Yaskawa INFORM job: KRIS5(-224_-90).JBI

/JOB
//NAME KRIS5(-224_-90)
//POS
///NPOS 254,254,254,14,0,0
///TOOL 0
///POSTYPE PULSE
///PULSE
C00000=126,-73357,-105376,-18827,72039,-77556
C00001=35778,-73357,-105376,-18827,72039,-77556
C00002=13505,189291,121101,-6814,55937,-83682
C00003=119958,189291,121101,-6814,55937,-83682
C00004=119958,189291,121101,-6814,55937,-83682
C00005=119958,189291,121101,-6814,96257,-82158
C00006=69507,150313,105301,-6814,81918,-83682
C00007=72199,118597,79738,-6814,91004,-83682
C00008=-14837,117754,79738,-6814,76523,-83682
C00009=-41681,102292,47908,-7222,67797,-83732
C00010=-106120,216,-72664,-1265,72875,-87293
C00011=-133015,-103640,-65816,3996,83698,-82063
C00012=-132086,-97485,-64003,4135,58701,-800
C00013=-131334,-97837,-53111,16599,61159,17527
C00014=-132395,-95402,-50215,16816,60857,17080
C00015=-132416,-94549,-48691,16897,60382,16996
C00016=-132416,-94725,-48971,16883,60461,17009
C00017=-132279,-93851,-48637,16827,60667,17094
C00018=-132382,-95256,-50220,16811,60927,17097
C00019=-94304,-90108,-48639,9529,56492,31191
C00020=-93667,-91692,-48976,9441,55822,31379
C00021=-93667,-90817,-47524,9489,55384,31339
C00022=-93667,-90990,-47811,9479,55470,31347
C00023=-93978,-90150,-47514,9528,55751,31249
C00024=-93593,-92158,-49496,9416,55894,31412
C00025=-118370,-114314,-60072,-4758,57984,4074
C00026=-118524,-103625,-49497,-4790,56962,4061
C00027=-114721,-103695,-48891,-5314,56776,5470
C00028=-114721,-102430,-47073,-5343,56310,5496
C00029=-114721,-103093,-48027,-5328,56554,5483
C00030=-114967,-100720,-47370,-5249,57351,5352
C00031=-114746,-103713,-49188,-5301,56945,5454
C00032=-161548,-94752,-46532,1465,58857,-11790
C00033=-161391,-93932,-45538,1444,58664,-11736
C00034=-161391,-92965,-44024,1450,58232,-11741
C00035=-161391,-93332,-44604,1446,58395,-11738
C00036=-160555,-92069,-44187,1319,58776,-11425
C00037=-161970,-95177,-46431,1528,58581,-11948
C00038=-123580,-122537,-67579,3227,57871,938
C00039=-106734,-120076,-67764,3834,76101,81400
C00040=-113343,-108186,-55340,6658,74419,78596
C00041=-116418,-106590,-51558,6363,73154,77529
C00042=-116418,-104744,-48943,6384,72498,77494
C00043=-116380,-105629,-49629,6389,72465,77504
C00044=-116257,-107112,-50007,6421,71928,77514
C00045=-116461,-105924,-51247,6354,73311,77523
C00046=-177893,-84927,-44498,-1145,82347,57715
C00047=-179150,-83983,-43048,-1323,81921,57309
C00048=-179150,-83213,-41718,-1324,81495,57312
C00049=-179506,-83879,-42356,-1373,81537,57197
C00050=-180639,-85061,-42804,-1534,81185,56832
C00051=-178742,-84413,-44413,-1264,82541,57436
C00052=-157426,-103778,-56504,-18034,71381,67764
C00053=-179018,-125046,-61555,-19353,59393,62032
C00054=-201764,-123429,-46759,-27362,51615,57091
C00055=-216699,-125747,-41034,-29303,43431,53713
C00056=-223595,-123281,-39482,-28787,41870,51323
C00057=-223595,-121879,-37858,-28937,41624,51414
C00058=-224642,-122442,-38457,-28819,41415,51031
C00059=-231128,-122675,-38460,-28269,39614,48820
C00060=-216121,-124277,-41147,-28911,44311,53639
C00061=-174045,-135981,-43542,-9522,59385,60566
C00062=-179227,-135331,-42329,-10713,58512,59173
C00063=-179227,-133640,-40520,-10741,58272,59200
C00064=-182821,-134437,-41073,-11535,57851,58216
C00065=-179482,-136401,-40870,-12350,56205,59776
C00066=-174986,-134999,-42396,-9751,59106,60326
C00067=-192579,-111155,-68057,-11776,89768,52211
C00068=-192579,-150013,-128024,-12422,106350,50582
C00069=-192579,-150013,-128024,-12422,106350,50582
C00070=-146460,-104346,-58758,-87,67702,67205
C00071=-164209,-65583,-26034,21815,71119,57818
C00072=-160784,-56678,-17427,19311,72734,59677
C00073=-160784,-55800,-15803,19364,72216,59591
C00074=-160784,-56161,-16471,19342,72429,59626
C00075=-161501,-57622,-17209,19332,72308,59354
C00076=-161057,-57134,-17514,19312,72624,59563
C00077=-152208,-64015,-24131,-4423,60929,65240
C00078=-158565,-56834,-16283,-17563,54636,65565
C00079=-158634,-56485,-15450,-17619,54304,65595
C00080=-158634,-55689,-13998,-17723,53845,65677
C00081=-158634,-56107,-14758,-17668,54088,65634
C00082=-159362,-57650,-15531,-17581,53638,65416
C00083=-158545,-56955,-16569,-17543,54755,65553
C00084=-153862,-55889,-14608,-19552,57702,67145
C00085=-161967,-50816,-11959,-18037,56866,64094
C00086=-148778,-72271,-33118,-3072,66412,73509
C00087=-145329,-64024,-24024,1262,65470,74080
C00088=-145576,-63687,-22619,1286,64785,73988
C00089=-134913,-66628,-23946,545,63974,77722
C00090=-140439,-69539,-27498,-3274,63016,76460
C00091=-160835,-97860,-53381,12033,68838,69115
C00092=-160835,-137865,-129483,11388,94610,71530
C00093=-160835,-137865,-129483,11388,94610,71530
C00094=-156474,-127565,-44757,-2910,70220,64434
C00095=-200400,-122534,-38487,-14714,65217,52406
C00096=-157255,-128893,-38327,-3230,65571,64341
C00097=-155117,-128273,-42851,-2556,68728,64843
C00098=-203941,-125612,-47386,-17033,60196,51476
C00099=-217380,-123179,-43051,-18833,56471,47671
C00100=-225173,-113450,-41869,-18656,59065,44558
C00101=-210006,-127688,-62340,-21133,60882,50691
C00102=-151947,-137880,-59984,-18934,60198,71208
C00103=-172289,-133022,-54384,-20839,55239,65166
C00104=-193729,-125214,-53607,-20379,54041,57625
C00105=-164056,-137190,-60910,-19878,58686,67360
C00106=-150051,-141583,-60664,6297,64762,70599
C00107=-159353,-138850,-55788,4675,63682,67765
C00108=-109486,-140583,-55786,12990,58412,82468
C00109=-146734,-145146,-63036,476,61954,73241
C00110=-164064,-147455,-64185,5609,61717,65893
C00111=-130860,-150279,-64151,-6173,30547,-11978
C00112=-130699,-138436,-62316,-8488,41278,7321
C00113=-138396,-134261,-59583,-6230,41150,4044
C00114=-146304,-133241,-59395,-3834,41140,659
C00115=-196433,-111576,-55328,9452,51613,-19605
C00116=-199673,-107900,-54372,9975,53256,-20719
C00117=-157623,-145161,-70844,16233,47931,-22606
C00118=-146088,-147027,-75251,-2759,46017,-11090
C00119=-148965,-131378,-70216,5109,51973,-19890
C00120=-151655,-124776,-64937,5631,52279,-20912
C00121=-97766,-126605,-65377,-5657,51601,-38
C00122=-113047,-122953,-63629,11912,53210,-15201
C00123=-135985,-140300,-81773,-1079,56771,-13995
C00124=-119711,-181360,-121572,-24950,66300,4723
C00125=-119711,-181360,-121572,-24950,66300,4723
C00126=-119711,-181360,-135603,-24950,39029,4723
C00127=-119711,-181360,-135603,-24950,39029,4723
C00128=-67118,-136665,-130676,-31892,63753,-5674
C00129=-38158,-160025,-136084,-39080,61805,-7690
C00130=-9060,-155984,-136090,-36075,61852,-27249
C00131=-9060,-155984,-136090,-36075,61852,-27249
C00132=35778,-73357,-105376,-18827,72039,-77556
C00133=35778,-73357,-105376,-18827,72039,-77556
C00134=121972,-60692,-66036,-23906,48760,-72917
C00135=121972,-63565,-66036,-13351,77444,-72917
C00136=129591,-43667,-50342,-15164,79318,-70462
C00137=130771,-42548,-47635,-15485,78487,-69942
C00138=130771,-42433,-46435,-15519,77830,-69855
C00139=130771,-42462,-46698,-15512,77973,-69874
C00140=130863,-43770,-47499,-15542,77817,-69821
C00141=130778,-42642,-47800,-15485,78538,-69942
C00142=106693,-40989,-47922,8584,79047,-76853
C00143=112828,-42305,-46652,18628,77879,-74099
C00144=112812,-42485,-45632,18678,77199,-74213
C00145=112812,-42347,-44543,18719,76632,-74301
C00146=112812,-42371,-44724,18712,76726,-74286
C00147=112739,-43676,-45526,18741,76573,-74337
C00148=112812,-42502,-45763,18675,77269,-74201
C00149=101589,-42073,-44271,32201,81327,-76893
C00150=104782,-94542,-85411,8339,74693,-77861
C00151=98731,-154827,-131308,9878,72678,-80158
C00152=98731,-154827,-131308,9878,72678,-80158
C00153=98731,-154827,-131308,9878,72678,-80158
C00154=141095,-137804,-121947,-4358,90462,-65341
C00155=171917,-153174,-112370,11397,78411,-54227
C00156=161217,-131665,-70261,12334,69937,-72545
C00157=174549,-127796,-65649,13485,67177,-68393
C00158=174549,-127096,-64796,13501,67016,-68412
C00159=175103,-127678,-65106,13549,66829,-68247
C00160=177071,-128966,-65326,13732,66020,-67678
C00161=174857,-128407,-66166,13506,67137,-68294
C00162=119665,-139437,-69480,-2305,70174,-83829
C00163=115014,-139487,-68249,-3034,69258,-85255
C00164=115014,-138034,-66654,-3036,69023,-85251
C00165=115014,-138331,-66981,-3035,69072,-85252
C00166=114723,-139907,-67140,-3094,68351,-85324
C00167=115018,-139674,-68474,-3029,69299,-85257
C00168=133085,-142772,-85485,-9589,79895,-78262
C00169=147328,-101232,-68657,-6996,92182,-74369
C00170=147006,-101545,-68639,-7054,91983,-74466
C00171=147006,-100879,-67432,-7052,91586,-74442
C00172=147006,-101065,-67769,-7053,91697,-74449
C00173=147583,-102934,-68401,-6943,91179,-74226
C00174=147081,-102142,-69356,-7044,92123,-74447
C00175=147950,-101609,-70952,8097,88078,-75282
C00176=157576,-95864,-68459,12752,86818,-72346
C00177=156860,-97500,-68064,12706,85871,-72691
C00178=156860,-96727,-66558,12711,85355,-72743
C00179=156860,-96921,-66934,12710,85484,-72730
C00180=157281,-97944,-67300,12748,85127,-72622
C00181=156374,-96868,-68790,12661,86704,-72773
C00182=143601,-106428,-78314,14904,88558,-77172
C00183=127839,-150907,-89343,18520,59767,-2936
C00184=132953,-138286,-79588,18019,59168,-1112
C00185=132445,-134119,-77799,17881,60264,-1120
C00186=132445,-132790,-76194,17931,59971,-1169
C00187=132445,-133640,-77222,17899,60159,-1137
C00188=131844,-130575,-76601,17754,61419,-1152
C00189=132709,-135969,-78749,17920,59858,-1088
C00190=132709,-135969,-78749,17920,59858,-1088
C00191=133237,-133582,-77709,17771,60311,-813
C00192=133237,-132259,-76100,17822,60018,-862
C00193=133237,-133036,-77045,17790,60191,-833
C00194=132722,-130580,-76544,17679,61206,-860
C00195=133601,-135952,-78909,17817,59782,-764
C00196=137036,-152242,-93003,17434,59376,467
C00197=169243,-109593,-79824,10807,67311,13542
C00198=171175,-102665,-75578,10363,67991,14312
C00199=170805,-101212,-73726,10463,67653,14148
C00200=170862,-101553,-74246,10441,67791,14177
C00201=169638,-99396,-73478,10634,68576,13802
C00202=171444,-103812,-77126,10284,68320,14438
C00203=136397,-123843,-83260,16295,67754,1500
C00204=137610,-120762,-80923,16148,67657,1933
C00205=137610,-119800,-79482,16191,67278,1880
C00206=137610,-120155,-80016,16174,67419,1899
C00207=137149,-117853,-79370,16140,68265,1848
C00208=137641,-121031,-81151,16144,67652,1943
C00209=135723,-130259,-80370,16559,56530,-240
C00210=176261,-108549,-74486,4912,58599,15900
C00211=180294,-103817,-72927,3633,59858,17504
C00212=168665,-137799,-89808,-4146,59076,16982
C00213=123783,-160681,-93004,13605,53968,-5410
C00214=114289,-158327,-83543,18281,44367,-10903
C00215=112815,-148174,-76256,18649,44789,-11465
C00216=188513,-127316,-73062,-7691,48720,21028
C00217=144715,-156700,-84216,13741,41290,797
C00218=138595,-119710,-81860,11603,79358,-76249
C00219=128675,-119099,-77606,11247,78465,-79723
C00220=133172,-119935,-74704,11559,75678,-78452
C00221=148695,-115278,-73215,11975,74934,-73204
C00222=145477,-116946,-76010,11872,76242,-74183
C00223=118816,-123903,-80121,-1281,78355,-81709
C00224=118014,-121625,-79522,-1328,79146,-81986
C00225=118504,-121794,-76164,-1305,76999,-81797
C00226=102382,-119997,-75746,-2266,77315,-87170
C00227=105330,-119244,-77878,-2083,79093,-86218
C00228=162093,-150282,-87461,-2658,71578,-66661
C00229=166503,-138624,-71158,-2287,67662,-65156
C00230=179660,-135656,-67070,1269,68997,-61418
C00231=154661,-142850,-67869,-2091,65690,-69226
C00232=147658,-138985,-70969,-2940,69389,-71507
C00233=167439,-135845,-70174,10586,65898,-66819
C00234=178556,-129130,-68304,14923,64423,-63985
C00235=183886,-128755,-65124,15213,61825,-62470
C00236=196612,-117976,-62765,14547,63647,-57713
C00237=190496,-117937,-66630,14420,66991,-59459
C00238=164740,-137810,-91614,20635,72894,-68588
C00239=164740,-137810,-91614,20635,72894,-68588
C00240=149447,-191890,-120181,21381,67024,-75156
C00241=149584,-192173,-120256,21405,66899,-75131
C00242=149584,-192173,-120256,21405,66899,-75131
C00243=135403,-47660,-52742,-16492,79886,-68488
C00244=133869,-36074,-43092,-15398,83056,-69397
C00245=126709,-37877,-44252,-14086,81561,-71713
C00246=124826,-51246,-53710,3634,72889,-70409
C00247=133954,-36259,-45628,1970,82055,-67034
C00248=132496,-35589,-44772,9764,81728,-66873
C00249=132387,-34090,-41818,9809,80707,-66990
C00250=136286,-32546,-39519,12831,78784,-65567
C00251=131832,-52683,-49405,33204,65462,-69826
C00252=109380,-75662,-60137,33198,63885,-64520
C00253=9054,-143647,-113334,-5954,77551,-79151
BC00000=192636,515545,1075136
BC00001=85474,515545,1075136
BC00002=85474,515545,1075136
BC00003=388258,515545,1075136
BC00004=388258,132939,1075136
BC00005=388258,132939,1075136
BC00006=266781,91691,1075136
BC00007=245343,24956,1075136
BC00008=171885,-116810,981693
BC00009=147620,-163639,1066245
BC00010=282408,-168564,1075136
BC00011=324871,12764,1075136
BC00012=324871,12764,1033476
BC00013=324871,12764,1033476
BC00014=324871,12764,1033476
BC00015=324871,12764,1033476
BC00016=324871,12764,1033476
BC00017=324871,12764,1033476
BC00018=324871,12764,1033472
BC00019=324871,12764,1033472
BC00020=324871,12764,1033472
BC00021=324871,12764,1033472
BC00022=324871,12764,1033472
BC00023=324871,12764,1033472
BC00024=324871,12764,1033472
BC00025=324871,12764,1033476
BC00026=324871,12764,1033476
BC00027=324871,12764,1033476
BC00028=324871,12764,1033476
BC00029=324871,12764,1033476
BC00030=324871,12764,1033476
BC00031=324871,12764,1033476
BC00032=324871,12764,1033476
BC00033=324871,12764,1033476
BC00034=324871,12764,1033476
BC00035=324871,12764,1033476
BC00036=324871,12764,1033476
BC00037=324871,12764,1033476
BC00038=324871,12764,1033476
BC00039=324871,42664,1033476
BC00040=324871,42664,1033476
BC00041=324871,42664,1033476
BC00042=324871,42664,1033476
BC00043=324871,42664,1033476
BC00044=324871,42664,1033476
BC00045=324871,42664,1033476
BC00046=324871,42664,1033476
BC00047=324871,42664,1033476
BC00048=324871,42664,1033476
BC00049=324871,42664,1033476
BC00050=324871,42664,1033476
BC00051=324871,42664,1033476
BC00052=324871,42664,1033476
BC00053=324871,42664,1033476
BC00054=324871,70402,1033476
BC00055=324871,70402,1033476
BC00056=324871,70402,1033476
BC00057=324871,70402,1033476
BC00058=324871,70402,1033476
BC00059=324871,70402,1033476
BC00060=324871,70402,1033476
BC00061=341363,70402,1033476
BC00062=341363,70402,1033476
BC00063=341363,70402,1033476
BC00064=341363,70402,1033476
BC00065=341363,70402,1033476
BC00066=341363,70402,1033476
BC00067=365604,67759,1033476
BC00068=365604,67759,1033476
BC00069=365604,-100317,1033476
BC00070=365604,-100317,1028280
BC00071=365604,-100317,1028280
BC00072=365604,-100317,1028280
BC00073=365604,-100317,1028280
BC00074=365604,-100317,1028280
BC00075=365604,-100317,1028280
BC00076=365604,-100317,1028280
BC00077=365604,-100317,1028280
BC00078=365604,-100317,1028280
BC00079=365604,-100317,1028280
BC00080=365604,-100317,1028280
BC00081=365604,-100317,1028280
BC00082=365604,-100317,1028280
BC00083=365604,-100317,1028280
BC00084=365604,-100317,1028280
BC00085=365604,-100317,1028280
BC00086=365604,-100317,1028280
BC00087=365604,-100317,1028280
BC00088=365604,-100317,1028280
BC00089=365604,-100317,1028280
BC00090=365604,-100317,1028280
BC00091=365604,-100317,1028280
BC00092=365604,-100317,1028280
BC00093=365604,-13875,1028280
BC00094=341538,67759,1033476
BC00095=341538,67759,1033476
BC00096=341538,67759,1033476
BC00097=341538,67759,1033476
BC00098=311299,64812,1025982
BC00099=311299,64812,1025982
BC00100=311299,64812,1025982
BC00101=318665,67846,1021463
BC00102=323021,86344,1018791
BC00103=323021,86344,1018791
BC00104=323021,86344,1018791
BC00105=323021,86344,1018791
BC00106=323021,86344,1018791
BC00107=323021,86344,1018791
BC00108=323021,86344,1018791
BC00109=323021,86344,1018791
BC00110=320650,86344,1061699
BC00111=320650,38724,1061699
BC00112=348099,38724,988490
BC00113=348099,38724,988490
BC00114=348099,38724,988490
BC00115=348099,38724,988490
BC00116=348099,38724,988490
BC00117=348099,38724,988490
BC00118=348099,38724,988490
BC00119=348099,38724,988490
BC00120=348099,38724,988490
BC00121=348099,38724,988490
BC00122=348099,38724,988490
BC00123=335935,44126,978638
BC00124=317547,52292,963745
BC00125=357240,-13468,1061786
BC00126=340345,-44387,1068891
BC00127=340345,-123490,1068891
BC00128=331767,-1766,1070081
BC00129=326806,106778,1070769
BC00130=344384,299723,1072198
BC00131=248648,436131,1072198
BC00132=295310,515545,1075136
BC00133=295310,515545,1075136
BC00134=295310,513263,813287
BC00135=335993,429318,731212
BC00136=335993,429318,731212
BC00137=335993,429318,731212
BC00138=335993,429318,731212
BC00139=335993,429318,731212
BC00140=335993,429318,731212
BC00141=335993,429318,731212
BC00142=292293,429318,731212
BC00143=292293,429318,731212
BC00144=292293,429318,731212
BC00145=292293,429318,731212
BC00146=292293,429318,731212
BC00147=292293,429318,731212
BC00148=292293,429318,731212
BC00149=292293,429318,731212
BC00150=292293,429318,731212
BC00151=292293,429318,979834
BC00152=314373,292172,979834
BC00153=314373,275872,695664
BC00154=349600,266255,695664
BC00155=349600,243768,695664
BC00156=318481,229664,891298
BC00157=318481,229664,891297
BC00158=318481,229664,891297
BC00159=318481,229664,891297
BC00160=318481,229664,891297
BC00161=318481,229664,891297
BC00162=333041,229664,891297
BC00163=333041,229664,891297
BC00164=333041,229664,891297
BC00165=333041,229664,891297
BC00166=333041,229664,891297
BC00167=333041,229664,891297
BC00168=347990,229664,891297
BC00169=347990,229664,891297
BC00170=347990,229664,891297
BC00171=347990,229664,891297
BC00172=347990,229664,891297
BC00173=347990,229664,891297
BC00174=347990,229664,891297
BC00175=347990,229664,891297
BC00176=331824,229664,891297
BC00177=331824,229664,891297
BC00178=331824,229664,891297
BC00179=331824,229664,891297
BC00180=331824,229664,891297
BC00181=331824,229664,891297
BC00182=317379,229664,891297
BC00183=317379,229664,891297
BC00184=317379,229664,891297
BC00185=317379,229664,891297
BC00186=317379,229664,891297
BC00187=317379,229664,891297
BC00188=317379,229664,891297
BC00189=317379,229664,891297
BC00190=361118,229664,891297
BC00191=361118,229664,891297
BC00192=361118,229664,891297
BC00193=361118,229664,891297
BC00194=361118,229664,891297
BC00195=361118,229664,891297
BC00196=317379,229664,891297
BC00197=317379,229664,891297
BC00198=317379,229664,891297
BC00199=317379,229664,891297
BC00200=317379,229664,891297
BC00201=317379,229664,891297
BC00202=317379,229664,891297
BC00203=317379,229664,891297
BC00204=317379,229664,891297
BC00205=317379,229664,891297
BC00206=317379,229664,891297
BC00207=317379,229664,891297
BC00208=317379,229664,891297
BC00209=317379,229664,891297
BC00210=317379,229664,891297
BC00211=317379,229664,891297
BC00212=326050,229664,891296
BC00213=343081,229663,891294
BC00214=340508,229663,891294
BC00215=343081,229663,891294
BC00216=343081,229663,891294
BC00217=323801,229663,891294
BC00218=310311,229663,891294
BC00219=310311,229663,891294
BC00220=310311,229663,891294
BC00221=310311,229663,891294
BC00222=310311,229663,891294
BC00223=310311,229663,891290
BC00224=327326,229663,891290
BC00225=327326,229663,891290
BC00226=327326,229663,891290
BC00227=327326,229663,891290
BC00228=351185,229663,891290
BC00229=351185,229663,891290
BC00230=351185,229663,891290
BC00231=351185,229663,891290
BC00232=351185,229663,891290
BC00233=335351,229663,891290
BC00234=335351,229663,891290
BC00235=335351,229663,891290
BC00236=335351,229663,891290
BC00237=335351,229663,891290
BC00238=335351,229663,891290
BC00239=352732,229663,1069777
BC00240=352732,229663,1069777
BC00241=352732,347909,1069777
BC00242=352732,347909,743295
BC00243=335993,429318,731212
BC00244=335993,429318,731212
BC00245=335993,429318,731212
BC00246=335994,429318,731211
BC00247=335994,429318,731211
BC00248=328432,429318,731211
BC00249=328432,429318,731211
BC00250=328432,429318,731211
BC00251=335994,429318,731211
BC00252=361465,487090,979283
BC00253=361465,516139,979283
EC00000=1986524,372644
EC00001=1986524,372644
EC00002=1986524,372644
EC00003=1986524,372644
EC00004=1986524,372644
EC00005=1986524,372644
EC00006=1986524,372644
EC00007=1986524,372644
EC00008=1986524,372644
EC00009=1986524,372644
EC00010=1986524,372644
EC00011=1986524,372644
EC00012=1986524,372644
EC00013=1986524,372644
EC00014=1986524,372644
EC00015=1986524,372644
EC00016=1986524,372644
EC00017=1986524,372644
EC00018=1986524,372643
EC00019=1986524,372643
EC00020=1986524,372643
EC00021=1986524,372643
EC00022=1986524,372643
EC00023=1986524,372643
EC00024=1986524,372643
EC00025=1986524,372644
EC00026=1986524,372644
EC00027=1986524,372644
EC00028=1986524,372644
EC00029=1986524,372644
EC00030=1986524,372644
EC00031=1986524,372644
EC00032=1986524,372644
EC00033=1986524,372644
EC00034=1986524,372644
EC00035=1986524,372644
EC00036=1986524,372644
EC00037=1986524,372644
EC00038=1986524,372644
EC00039=1986524,372644
EC00040=1986524,372644
EC00041=1986524,372644
EC00042=1986524,372644
EC00043=1986524,372644
EC00044=1986524,372644
EC00045=1986524,372644
EC00046=1986524,372644
EC00047=1986524,372644
EC00048=1986524,372644
EC00049=1986524,372644
EC00050=1986524,372644
EC00051=1986524,372644
EC00052=1986524,372644
EC00053=1986524,372644
EC00054=1986524,372644
EC00055=1986524,372644
EC00056=1986524,372644
EC00057=1986524,372644
EC00058=1986524,372644
EC00059=1986524,372644
EC00060=1986524,372644
EC00061=1986524,372644
EC00062=1986524,372644
EC00063=1986524,372644
EC00064=1986524,372644
EC00065=1986524,372644
EC00066=1986524,372644
EC00067=1986524,372644
EC00068=1986524,372644
EC00069=1986524,372644
EC00070=1986525,372644
EC00071=1986525,372644
EC00072=1986525,372644
EC00073=1986525,372644
EC00074=1986525,372644
EC00075=1986525,372644
EC00076=1986525,372644
EC00077=1986525,372644
EC00078=1986525,372644
EC00079=1986525,372644
EC00080=1986525,372644
EC00081=1986525,372644
EC00082=1986525,372644
EC00083=1986525,372644
EC00084=1986525,372644
EC00085=1986525,372644
EC00086=1986525,372644
EC00087=1986525,372644
EC00088=1986525,372644
EC00089=1986525,372644
EC00090=1986525,372644
EC00091=1986525,372644
EC00092=1986525,372644
EC00093=1986525,372644
EC00094=1986524,372644
EC00095=1986524,372644
EC00096=1986524,372644
EC00097=1986524,372644
EC00098=1986524,372644
EC00099=1986524,372644
EC00100=1986524,372644
EC00101=1986524,372644
EC00102=1986524,372644
EC00103=1986524,372644
EC00104=1986524,372644
EC00105=1986524,372644
EC00106=1986524,372644
EC00107=1986524,372644
EC00108=1986524,372644
EC00109=1986524,372644
EC00110=1986524,372644
EC00111=1986524,372644
EC00112=1986524,372644
EC00113=1986524,372644
EC00114=1986524,372644
EC00115=1986524,372644
EC00116=1986524,372644
EC00117=1986524,372644
EC00118=1986524,372644
EC00119=1986524,372644
EC00120=1986524,372644
EC00121=1986524,372644
EC00122=1986524,372644
EC00123=1986524,372644
EC00124=1986524,372644
EC00125=1986524,372644
EC00126=1986524,372644
EC00127=1986524,372644
EC00128=1924386,269829
EC00129=1888448,210364
EC00130=1813786,86826
EC00131=1784464,86826
EC00132=1660311,-167120
EC00133=1153659,-722953
EC00134=1144025,-740308
EC00135=1144025,-740308
EC00136=1144025,-740308
EC00137=1144025,-740308
EC00138=1144025,-740308
EC00139=1144025,-740308
EC00140=1144025,-740308
EC00141=1144025,-740308
EC00142=1144025,-740308
EC00143=1144025,-740308
EC00144=1144025,-740308
EC00145=1144025,-740308
EC00146=1144025,-740308
EC00147=1144025,-740308
EC00148=1144025,-740308
EC00149=1144025,-740308
EC00150=1144025,-740308
EC00151=1144025,-740308
EC00152=1144025,-740308
EC00153=1144025,-740308
EC00154=1144025,-740308
EC00155=1144025,-740308
EC00156=1144025,-740308
EC00157=1144024,-740308
EC00158=1144024,-740308
EC00159=1144024,-740308
EC00160=1144024,-740308
EC00161=1144024,-740308
EC00162=1144024,-740308
EC00163=1144024,-740308
EC00164=1144024,-740308
EC00165=1144024,-740308
EC00166=1144024,-740308
EC00167=1144024,-740308
EC00168=1144023,-740308
EC00169=1144023,-740308
EC00170=1144023,-740308
EC00171=1144023,-740308
EC00172=1144023,-740308
EC00173=1144023,-740308
EC00174=1144023,-740308
EC00175=1144023,-740308
EC00176=1144023,-740308
EC00177=1144023,-740308
EC00178=1144023,-740308
EC00179=1144023,-740308
EC00180=1144023,-740308
EC00181=1144023,-740308
EC00182=1144023,-740308
EC00183=1144023,-740308
EC00184=1144023,-740308
EC00185=1144023,-740308
EC00186=1144023,-740308
EC00187=1144023,-740308
EC00188=1144023,-740308
EC00189=1144023,-740308
EC00190=1144023,-740308
EC00191=1144023,-740308
EC00192=1144023,-740308
EC00193=1144023,-740308
EC00194=1144023,-740308
EC00195=1144023,-740308
EC00196=1144023,-740308
EC00197=1144023,-740308
EC00198=1144023,-740308
EC00199=1144023,-740308
EC00200=1144023,-740308
EC00201=1144023,-740308
EC00202=1144023,-740308
EC00203=1144023,-740308
EC00204=1144023,-740308
EC00205=1144023,-740308
EC00206=1144023,-740308
EC00207=1144023,-740308
EC00208=1144023,-740308
EC00209=1144023,-740308
EC00210=1144023,-740308
EC00211=1144023,-740308
EC00212=1144021,-740308
EC00213=1144019,-740308
EC00214=1144019,-740308
EC00215=1144019,-740308
EC00216=1144019,-740308
EC00217=1144019,-740308
EC00218=1144019,-740308
EC00219=1144019,-740308
EC00220=1144019,-740308
EC00221=1144019,-740308
EC00222=1144019,-740308
EC00223=1144018,-740308
EC00224=1144018,-740308
EC00225=1144018,-740308
EC00226=1144018,-740308
EC00227=1144018,-740308
EC00228=1144018,-740308
EC00229=1144018,-740308
EC00230=1144018,-740308
EC00231=1144018,-740308
EC00232=1144018,-740308
EC00233=1144018,-740308
EC00234=1144018,-740308
EC00235=1144018,-740308
EC00236=1144018,-740308
EC00237=1144018,-740308
EC00238=1144018,-740308
EC00239=1144018,-740308
EC00240=1144018,-740308
EC00241=1144018,-740308
EC00242=1144018,-740308
EC00243=1144025,-740308
EC00244=1144025,-740308
EC00245=1144025,-740308
EC00246=1144023,-740309
EC00247=1144023,-740309
EC00248=1144023,-740309
EC00249=1144023,-740309
EC00250=1144023,-740309
EC00251=1144023,-740309
EC00252=1144023,-740309
EC00253=1144023,-740309
///POSTYPE BASE
///RECTAN
///RCONF 0,0,0,0,1,0,0,0,0,0,0,0,0,0,0,0,0,0,0,0,0,0,0,0
P00006=2.006,1.622,-0.565,0.0000,0.0000,0.0000
P00021=0.073,2.058,-0.109,0.0000,0.0000,0.0000
P00022=2.006,1.622,-0.565,0.0000,0.0000,0.0000
///RCONF 0,0,0,0,0,0,0,0,0,0,0,0,0,0,0,0,0,0,0,0,0,0,0,0
P00023=-2.957,-4.083,2.762,0.0000,0.0000,0.0000
P00024=-1.466,-0.226,-0.419,0.0000,0.0000,0.0000
P00025=3.643,0.007,-2.585,0.0000,0.0000,0.0000
P00026=2.644,0.055,-2.583,0.0000,0.0000,0.0000
P00027=2.278,0.099,-4.210,0.0000,0.0000,0.0000
P00028=-1.778,-0.182,-2.050,0.0000,0.0000,0.0000
P00029=1.749,4.006,-0.261,0.0000,0.0000,0.0000
P00030=-0.014,-0.768,0.131,0.0000,0.0000,0.0000
P00031=-0.170,0.039,-0.647,0.0000,0.0000,0.0000
P00032=-0.423,0.157,3.222,0.0000,0.0000,0.0000
P00033=0.854,-1.099,3.047,0.0000,0.0000,0.0000
//INST
///DATE 2024/10/31 15:24
///ATTR SC,RW
///GROUP1 RB1,BS1
///GROUP2 ST1
NOP
'010224 MUZYLO
MOVJ C00000 BC00000 VJ=100.00  +MOVJ EC00000 VJ=100.00
CALL JOB:CLEAN-R1_KM_NEW
MOVJ C00001 BC00001 VJ=100.00  +MOVJ EC00001 VJ=100.00
MOVJ C00002 BC00002 VJ=100.00  +MOVJ EC00002 VJ=100.00
MOVJ C00003 BC00003 VJ=70.00  +MOVJ EC00003 VJ=100.00
MOVJ C00004 BC00004 VJ=60.00  +MOVJ EC00004 VJ=100.00
MOVJ C00005 BC00005 VJ=100.00  +MOVJ EC00005 VJ=100.00
MOVJ C00006 BC00006 VJ=100.00  +MOVJ EC00006 VJ=100.00
MOVJ C00007 BC00007 VJ=100.00  +MOVJ EC00007 VJ=100.00
MOVJ C00008 BC00008 VJ=100.00  +MOVJ EC00008 VJ=100.00
MOVJ C00009 BC00009 VJ=100.00  +MOVJ EC00009 VJ=100.00
MOVJ C00010 BC00010 VJ=100.00  +MOVJ EC00010 VJ=100.00
MOVJ C00011 BC00011 VJ=100.00  +MOVJ EC00011 VJ=100.00
MOVJ C00012 BC00012 VJ=100.00  +MOVJ EC00012 VJ=100.00
MOVJ C00013 BC00013 VJ=100.00  +MOVJ EC00013 VJ=100.00
SFTOF3D
SMOVL C00014 BC00014 V=100.0  +MOVJ EC00014
SREFP 3 C00015 BC00015  +REFP EC00015
CALL JOB:SEARCH-R1-S13D
SET P032 P006
SFTON3D P032
SMOVL C00016 BC00016 V=100.0  +MOVJ EC00016
SREFP 3 C00017 BC00017  +REFP EC00017
CALL JOB:SEARCH-R1-S13D
SET P032 P006
SFTON3D P032
SMOVL C00018 BC00018 V=100.0  +MOVJ EC00018
SFTOF3D
SMOVL C00019 BC00019 V=250.0  +MOVJ EC00019
SMOVL C00020 BC00020 V=100.0  +MOVJ EC00020
SREFP 3 C00021 BC00021  +REFP EC00021
CALL JOB:SEARCH-R1-S13D
SET P033 P006
SFTON3D P033
SMOVL C00022 BC00022 V=100.0  +MOVJ EC00022
SREFP 3 C00023 BC00023  +REFP EC00023
CALL JOB:SEARCH-R1-S13D
SET P033 P006
SFTON3D P033
SMOVL C00024 BC00024 V=100.0  +MOVJ EC00024
SFTOF3D
SMOVL C00025 BC00025 V=250.0  +MOVJ EC00025
SMOVL C00026 BC00026 V=416.7  +MOVJ EC00026
SMOVL C00027 BC00027 V=100.0  +MOVJ EC00027
SREFP 3 C00028 BC00028  +REFP EC00028
CALL JOB:SEARCH-R1-S13D
SET P030 P006
SFTON3D P030
SMOVL C00029 BC00029 V=100.0  +MOVJ EC00029
SREFP 3 C00030 BC00030  +REFP EC00030
CALL JOB:SEARCH-R1-S13D
SET P030 P006
SFTON3D P030
SMOVL C00031 BC00031 V=100.0  +MOVJ EC00031
SFTOF3D
SMOVL C00032 BC00032 V=500.0  +MOVJ EC00032
SMOVL C00033 BC00033 V=100.0  +MOVJ EC00033
SREFP 3 C00034 BC00034  +REFP EC00034
CALL JOB:SEARCH-R1-S13D
SET P031 P006
SFTON3D P031
SMOVL C00035 BC00035 V=100.0  +MOVJ EC00035
SREFP 3 C00036 BC00036  +REFP EC00036
CALL JOB:SEARCH-R1-S13D
SET P031 P006
SFTON3D P031
SMOVL C00037 BC00037 V=100.0  +MOVJ EC00037
SFTOF3D
MOVJ C00038 BC00038 VJ=100.00  +MOVJ EC00038 VJ=100.00
MOVJ C00039 BC00039 VJ=100.00  +MOVJ EC00039 VJ=50.00
MOVJ C00040 BC00040 VJ=100.00  +MOVJ EC00040 VJ=50.00
SMOVL C00041 BC00041 V=100.0  +MOVJ EC00041
SREFP 3 C00042 BC00042  +REFP EC00042
CALL JOB:SEARCH-R1-S13D
SET P021 P006
SFTON3D P021
SMOVL C00043 BC00043 V=100.0  +MOVJ EC00043
SREFP 3 C00044 BC00044  +REFP EC00044
CALL JOB:SEARCH-R1-S13D
SET P021 P006
SFTON3D P021
SMOVL C00045 BC00045 V=100.0  +MOVJ EC00045
SFTOF3D
SMOVL C00046 BC00046 V=500.0  +MOVJ EC00046
SMOVL C00047 BC00047 V=100.0  +MOVJ EC00047
SREFP 3 C00048 BC00048  +REFP EC00048
CALL JOB:SEARCH-R1-S13D
SET P022 P006
SFTON3D P022
SMOVL C00049 BC00049 V=100.0  +MOVJ EC00049
SREFP 3 C00050 BC00050  +REFP EC00050
CALL JOB:SEARCH-R1-S13D
SET P022 P006
SFTON3D P022
SMOVL C00051 BC00051 V=100.0  +MOVJ EC00051
SFTOF3D
SMOVL C00052 BC00052 V=333.3  +MOVJ EC00052
SMOVL C00053 BC00053 V=666.7  +MOVJ EC00053
SMOVL C00054 BC00054 V=666.7  +MOVJ EC00054
SMOVL C00055 BC00055 V=333.3  +MOVJ EC00055
SMOVL C00056 BC00056 V=100.0  +MOVJ EC00056
SREFP 3 C00057 BC00057  +REFP EC00057
CALL JOB:SEARCH-R1-S13D
SET P024 P006
SFTON3D P024
SMOVL C00058 BC00058 V=100.0  +MOVJ EC00058
SREFP 3 C00059 BC00059  +REFP EC00059
CALL JOB:SEARCH-R1-S13D
SET P024 P006
SFTON3D P024
SMOVL C00060 BC00060 V=100.0  +MOVJ EC00060
SFTOF3D
SMOVL C00061 BC00061 V=500.0  +MOVJ EC00061
SMOVL C00062 BC00062 V=100.0  +MOVJ EC00062
SREFP 3 C00063 BC00063  +REFP EC00063
CALL JOB:SEARCH-R1-S13D
SET P025 P006
SFTON3D P025
SMOVL C00064 BC00064 V=100.0  +MOVJ EC00064
SREFP 3 C00065 BC00065  +REFP EC00065
CALL JOB:SEARCH-R1-S13D
SET P025 P006
SFTON3D P025
SMOVL C00066 BC00066 V=100.0  +MOVJ EC00066
SFTOF3D
MOVJ C00067 BC00067 VJ=50.00  +MOVJ EC00067 VJ=50.00
MOVJ C00068 BC00068 VJ=100.00  +MOVJ EC00068 VJ=50.00
MOVJ C00069 BC00069 VJ=100.00  +MOVJ EC00069 VJ=50.00
MOVJ C00070 BC00070 VJ=100.00  +MOVJ EC00070 VJ=50.00
MOVJ C00071 BC00071 VJ=100.00  +MOVJ EC00071 VJ=50.00
SMOVL C00072 BC00072 V=133.3  +MOVJ EC00072
SREFP 3 C00073 BC00073  +REFP EC00073
CALL JOB:SEARCH-R1-S13D
SET P027 P006
SFTON3D P027
SMOVL C00074 BC00074 V=100.0  +MOVJ EC00074
SREFP 3 C00075 BC00075  +REFP EC00075
CALL JOB:SEARCH-R1-S13D
SET P027 P006
SFTON3D P027
SMOVL C00076 BC00076 V=100.0  +MOVJ EC00076
SFTOF3D
SMOVL C00077 BC00077 V=416.7  +MOVJ EC00077
SMOVL C00078 BC00078 V=416.7  +MOVJ EC00078
SMOVL C00079 BC00079 V=100.0  +MOVJ EC00079
SREFP 3 C00080 BC00080  +REFP EC00080
CALL JOB:SEARCH-R1-S13D
SET P028 P006
SFTON3D P028
SMOVL C00081 BC00081 V=100.0  +MOVJ EC00081
SREFP 3 C00082 BC00082  +REFP EC00082
CALL JOB:SEARCH-R1-S13D
SET P028 P006
SFTON3D P028
SMOVL C00083 BC00083 V=100.0  +MOVJ EC00083
MACRO1 MJ#(0) ARGF14
'SPAWANIE 1CZ.
SMOVL C00084 BC00084 V=133.3  +MOVJ EC00084
ARCON
SMOVL C00085 BC00085 V=10.0  +MOVJ EC00085
ARCOF
SFTOF3D
SMOVL C00086 BC00086 V=250.0  +MOVJ EC00086
SMOVL C00087 BC00087 V=250.0  +MOVJ EC00087
SFTON3D P027
SMOVL C00088 BC00088 V=133.3  +MOVJ EC00088
ARCON
SMOVL C00089 BC00089 V=10.0  +MOVJ EC00089
ARCOF
SFTOF3D
SMOVL C00090 BC00090 V=133.3  +MOVJ EC00090
MOVJ C00091 BC00091 VJ=100.00  +MOVJ EC00091 VJ=50.00
MOVJ C00092 BC00092 VJ=100.00  +MOVJ EC00092 VJ=50.00
MOVJ C00093 BC00093 VJ=100.00  +MOVJ EC00093 VJ=100.00
MOVJ C00094 BC00094 VJ=100.00  +MOVJ EC00094 VJ=100.00
SFTON3D P025
SMOVL C00095 BC00095 V=133.3  +MOVJ EC00095
ARCON
SMOVL C00096 BC00096 V=10.0  +MOVJ EC00096
ARCOF
SFTOF3D
SMOVL C00097 BC00097 V=250.0  +MOVJ EC00097
SMOVL C00098 BC00098 V=666.7  +MOVJ EC00098
SFTON3D P024
SMOVL C00099 BC00099 V=133.3  +MOVJ EC00099
ARCON
SMOVL C00100 BC00100 V=10.0  +MOVJ EC00100
ARCOF
SFTOF3D
SMOVL C00101 BC00101 V=250.0  +MOVJ EC00101
SMOVL C00102 BC00102 V=416.7  +MOVJ EC00102
SFTON3D P022
SMOVL C00103 BC00103 V=133.3  +MOVJ EC00103
ARCON
SMOVL C00104 BC00104 V=10.0  +MOVJ EC00104
ARCOF
SFTOF3D
SMOVL C00105 BC00105 V=250.0  +MOVJ EC00105
SMOVL C00106 BC00106 V=500.0  +MOVJ EC00106
SFTON3D P021
SMOVL C00107 BC00107 V=133.3  +MOVJ EC00107
ARCON
SMOVL C00108 BC00108 V=10.0  +MOVJ EC00108
ARCOF
SFTOF3D
SMOVL C00109 BC00109 V=250.0  +MOVJ EC00109
MOVJ C00110 BC00110 VJ=100.00  +MOVJ EC00110 VJ=100.00
MOVJ C00111 BC00111 VJ=100.00  +MOVJ EC00111 VJ=100.00
MOVJ C00112 BC00112 VJ=80.00  +MOVJ EC00112 VJ=100.00
SFTON3D P030
SMOVL C00113 BC00113 V=133.3  +MOVJ EC00113
ARCON
SMOVL C00114 BC00114 V=8.3  +MOVJ EC00114
SFTON3D P031
SMOVL C00115 BC00115 V=8.3  +MOVJ EC00115
SMOVL C00116 BC00116 V=8.3  +MOVJ EC00116
ARCOF
SFTOF3D
SMOVL C00117 BC00117 V=250.0  +MOVJ EC00117
SMOVL C00118 BC00118 V=400.0  +MOVJ EC00118
SMOVL C00119 BC00119 V=400.0  +MOVJ EC00119
MACRO1 MJ#(0) ARGF9
SFTON3D P032
SMOVL C00120 BC00120 V=133.3  +MOVJ EC00120
ARCON
SFTON3D P033
SMOVL C00121 BC00121 V=10.0  +MOVJ EC00121
SMOVL C00122 BC00122 V=10.0  +MOVJ EC00122
ARCOF
SFTOF3D
SMOVL C00123 BC00123 V=500.0  +MOVJ EC00123
MOVJ C00124 BC00124 VJ=100.00  +MOVJ EC00124 VJ=30.00
MOVJ C00125 BC00125 VJ=100.00  +MOVJ EC00125 VJ=100.00
MOVJ C00126 BC00126 VJ=100.00  +MOVJ EC00126 VJ=100.00
MOVJ C00127 BC00127 VJ=100.00  +MOVJ EC00127 VJ=100.00
MOVJ C00128 BC00128 VJ=100.00  +MOVJ EC00128 VJ=100.00
MOVJ C00129 BC00129 VJ=100.00  +MOVJ EC00129 VJ=100.00
MOVJ C00130 BC00130 VJ=100.00  +MOVJ EC00130 VJ=100.00
MOVJ C00131 BC00131 VJ=30.00  +MOVJ EC00131 VJ=30.00
'DRUGA POZYCJA
MOVJ C00132 BC00132 VJ=100.00  +MOVJ EC00132 VJ=100.00
MOVJ C00133 BC00133 VJ=100.00  +MOVJ EC00133 VJ=100.00
CALL JOB:CLEAN-R1_KM_NEW
MOVJ C00134 BC00134 VJ=100.00  +MOVJ EC00134 VJ=100.00
MOVJ C00135 BC00135 VJ=100.00  +MOVJ EC00135 VJ=100.00
MOVJ C00136 BC00136 VJ=100.00  +MOVJ EC00136 VJ=100.00
SMOVL C00137 BC00137 V=100.0  +MOVJ EC00137
SREFP 3 C00138 BC00138  +REFP EC00138
CALL JOB:SEARCH-R1-S13D
SET P021 P006
SFTON3D P021
SMOVL C00139 BC00139 V=100.0  +MOVJ EC00139
SREFP 3 C00140 BC00140  +REFP EC00140
CALL JOB:SEARCH-R1-S13D
SET P021 P006
SFTON3D P021
SMOVL C00141 BC00141 V=100.0  +MOVJ EC00141
SFTOF3D
SMOVL C00142 BC00142 V=250.0  +MOVJ EC00142
SMOVL C00143 BC00143 V=333.3  +MOVJ EC00143
SMOVL C00144 BC00144 V=100.0  +MOVJ EC00144
SREFP 3 C00145 BC00145  +REFP EC00145
CALL JOB:SEARCH-R1-S13D
SET P023 P006
SFTON3D P023
SMOVL C00146 BC00146 V=100.0  +MOVJ EC00146
SREFP 3 C00147 BC00147  +REFP EC00147
CALL JOB:SEARCH-R1-S13D
SET P023 P006
SFTON3D P023
SMOVL C00148 BC00148 V=100.0  +MOVJ EC00148
SFTOF3D
SSFTOF
SFTOF
SMOVL C00149 BC00149 V=333.3  +MOVJ EC00149
SMOVL C00150 BC00150 V=333.3  +MOVJ EC00150
SMOVL C00151 BC00151 V=333.3  +MOVJ EC00151
MOVJ C00152 BC00152 VJ=100.00  +MOVJ EC00152 VJ=100.00
MOVJ C00153 BC00153 VJ=100.00  +MOVJ EC00153 VJ=100.00
MOVJ C00154 BC00154 VJ=100.00  +MOVJ EC00154 VJ=100.00
MOVJ C00155 BC00155 VJ=100.00  +MOVJ EC00155 VJ=100.00
SMOVL C00156 BC00156 V=333.3  +MOVJ EC00156
SMOVL C00157 BC00157 V=100.0  +MOVJ EC00157
SREFP 3 C00158 BC00158  +REFP EC00158
CALL JOB:SEARCH-R1-S13D
SET P024 P006
SFTON3D P024
SMOVL C00159 BC00159 V=100.0  +MOVJ EC00159
SREFP 3 C00160 BC00160  +REFP EC00160
CALL JOB:SEARCH-R1-S13D
SET P024 P006
SFTON3D P024
SMOVL C00161 BC00161 V=100.0  +MOVJ EC00161
SFTOF3D
SMOVL C00162 BC00162 V=333.3  +MOVJ EC00162
SMOVL C00163 BC00163 V=100.0  +MOVJ EC00163
SREFP 3 C00164 BC00164  +REFP EC00164
CALL JOB:SEARCH-R1-S13D
SET P026 P006
SFTON3D P026
SMOVL C00165 BC00165 V=100.0  +MOVJ EC00165
SREFP 3 C00166 BC00166  +REFP EC00166
CALL JOB:SEARCH-R1-S13D
SET P026 P006
SFTON3D P026
SMOVL C00167 BC00167 V=100.0  +MOVJ EC00167
SFTOF3D
MOVJ C00168 BC00168 VJ=100.00  +MOVJ EC00168 VJ=50.00
MOVJ C00169 BC00169 VJ=100.00  +MOVJ EC00169 VJ=50.00
SMOVL C00170 BC00170 V=100.0  +MOVJ EC00170
SREFP 3 C00171 BC00171  +REFP EC00171
CALL JOB:SEARCH-R1-S13D
SET P027 P006
SFTON3D P027
SMOVL C00172 BC00172 V=100.0  +MOVJ EC00172
SREFP 3 C00173 BC00173  +REFP EC00173
CALL JOB:SEARCH-R1-S13D
SET P027 P006
SFTON3D P027
SMOVL C00174 BC00174 V=100.0  +MOVJ EC00174
SFTOF3D
SMOVL C00175 BC00175 V=416.7  +MOVJ EC00175
SMOVL C00176 BC00176 V=416.7  +MOVJ EC00176
SMOVL C00177 BC00177 V=100.0  +MOVJ EC00177
SREFP 3 C00178 BC00178  +REFP EC00178
CALL JOB:SEARCH-R1-S13D
SET P029 P006
SFTON3D P029
SMOVL C00179 BC00179 V=100.0  +MOVJ EC00179
SREFP 3 C00180 BC00180  +REFP EC00180
CALL JOB:SEARCH-R1-S13D
SET P029 P006
SFTON3D P029
SMOVL C00181 BC00181 V=100.0  +MOVJ EC00181
MOVJ C00182 BC00182 VJ=100.00  +MOVJ EC00182 VJ=100.00
MOVJ C00183 BC00183 VJ=100.00  +MOVJ EC00183 VJ=100.00
MOVJ C00184 BC00184 VJ=100.00  +MOVJ EC00184 VJ=100.00
SMOVL C00185 BC00185 V=100.0  +MOVJ EC00185
SREFP 3 C00186 BC00186  +REFP EC00186
CALL JOB:SEARCH-R1-S13D
SET P030 P006
SFTON3D P030
SMOVL C00187 BC00187 V=100.0  +MOVJ EC00187
SREFP 3 C00188 BC00188  +REFP EC00188
CALL JOB:SEARCH-R1-S13D
SET P030 P006
SFTON3D P030
SMOVL C00189 BC00189 V=100.0  +MOVJ EC00189
SFTOF3D
SMOVL C00190 BC00190 V=500.0  +MOVJ EC00190
SMOVL C00191 BC00191 V=100.0  +MOVJ EC00191
SREFP 3 C00192 BC00192  +REFP EC00192
CALL JOB:SEARCH-R1-S13D
SET P031 P006
SFTON3D P031
SMOVL C00193 BC00193 V=100.0  +MOVJ EC00193
SREFP 3 C00194 BC00194  +REFP EC00194
CALL JOB:SEARCH-R1-S13D
SET P031 P006
SFTON3D P031
SMOVL C00195 BC00195 V=100.0  +MOVJ EC00195
SFTOF3D
SMOVL C00196 BC00196 V=500.0  +MOVJ EC00196
SMOVL C00197 BC00197 V=500.0  +MOVJ EC00197
SMOVL C00198 BC00198 V=100.0  +MOVJ EC00198
SREFP 3 C00199 BC00199  +REFP EC00199
CALL JOB:SEARCH-R1-S13D
SET P033 P006
SFTON3D P033
SMOVL C00200 BC00200 V=100.0  +MOVJ EC00200
SREFP 3 C00201 BC00201  +REFP EC00201
CALL JOB:SEARCH-R1-S13D
SET P033 P006
SFTON3D P033
SMOVL C00202 BC00202 V=100.0  +MOVJ EC00202
SFTOF3D
SMOVL C00203 BC00203 V=250.0  +MOVJ EC00203
SMOVL C00204 BC00204 V=100.0  +MOVJ EC00204
SREFP 3 C00205 BC00205  +REFP EC00205
CALL JOB:SEARCH-R1-S13D
SET P032 P006
SFTON3D P032
SMOVL C00206 BC00206 V=100.0  +MOVJ EC00206
SREFP 3 C00207 BC00207  +REFP EC00207
CALL JOB:SEARCH-R1-S13D
SET P032 P006
SFTON3D P032
SMOVL C00208 BC00208 V=100.0  +MOVJ EC00208
MACRO1 MJ#(0) ARGF14
SMOVL C00209 BC00209 V=166.7  +MOVJ EC00209
ARCON
SFTON3D P033
SMOVL C00210 BC00210 V=8.3  +MOVJ EC00210
SMOVL C00211 BC00211 V=8.3  +MOVJ EC00211
ARCOF
SFTOF3D
SMOVL C00212 BC00212 V=416.7  +MOVJ EC00212
SMOVL C00213 BC00213 V=416.7  +MOVJ EC00213
SMOVL C00214 BC00214 V=416.7  +MOVJ EC00214
SFTON3D P030
SMOVL C00215 BC00215 V=133.3  +MOVJ EC00215
ARCON
SFTON3D P031
SMOVL C00216 BC00216 V=8.3  +MOVJ EC00216
ARCOF
SFTOF3D
SMOVL C00217 BC00217 V=416.7  +MOVJ EC00217
MOVJ C00218 BC00218 VJ=100.00  +MOVJ EC00218 VJ=100.00
MOVJ C00219 BC00219 VJ=15.00  +MOVJ EC00219 VJ=100.00
SFTON3D P029
SMOVL C00220 BC00220 V=133.3  +MOVJ EC00220
ARCON
MOVL C00221 BC00221 V=10.0  +MOVJ EC00221 VJ=15.00
ARCOF
MOVJ C00222 BC00222 VJ=30.00  +MOVJ EC00222 VJ=15.00
SFTOF3D
SMOVL C00223 BC00223 V=500.0  +MOVJ EC00223
SMOVL C00224 BC00224 V=500.0  +MOVJ EC00224
SFTON3D P027
SMOVL C00225 BC00225 V=133.3  +MOVJ EC00225
ARCON
SMOVL C00226 BC00226 V=10.0  +MOVJ EC00226
ARCOF
SFTOF3D
SMOVL C00227 BC00227 V=250.0  +MOVJ EC00227
SMOVL C00228 BC00228 V=500.0  +MOVJ EC00228
SMOVL C00229 BC00229 V=500.0  +MOVJ EC00229
SFTON3D P026
SMOVL C00230 BC00230 V=133.3  +MOVJ EC00230
ARCON
SMOVL C00231 BC00231 V=10.0  +MOVJ EC00231
ARCOF
SFTOF3D
SMOVL C00232 BC00232 V=250.0  +MOVJ EC00232
SMOVL C00233 BC00233 V=500.0  +MOVJ EC00233
SMOVL C00234 BC00234 V=500.0  +MOVJ EC00234
SFTON3D P024
SMOVL C00235 BC00235 V=133.3  +MOVJ EC00235
ARCON
SMOVL C00236 BC00236 V=10.0  +MOVJ EC00236
ARCOF
SMOVL C00237 BC00237 V=250.0  +MOVJ EC00237
SFTOF3D
SMOVL C00238 BC00238 V=500.0  +MOVJ EC00238
SMOVL C00239 BC00239 V=500.0  +MOVJ EC00239
SMOVL C00240 BC00240 V=500.0  +MOVJ EC00240
SMOVL C00241 BC00241 V=500.0  +MOVJ EC00241
SMOVL C00242 BC00242 V=500.0  +MOVJ EC00242
SMOVL C00243 BC00243 V=500.0  +MOVJ EC00243
SFTON3D P021
SMOVL C00244 BC00244 V=133.3  +MOVJ EC00244
ARCON
SMOVL C00245 BC00245 V=10.0  +MOVJ EC00245
ARCOF
SFTOF3D
SMOVL C00246 BC00246 V=250.0  +MOVJ EC00246
SMOVL C00247 BC00247 V=250.0  +MOVJ EC00247
SMOVL C00248 BC00248 V=333.3  +MOVJ EC00248
SFTON3D P023
SMOVL C00249 BC00249 V=133.3  +MOVJ EC00249
ARCON
SMOVL C00250 BC00250 V=10.0  +MOVJ EC00250
ARCOF
SFTOF3D
SFTOF
SMOVL C00251 BC00251 V=250.0  +MOVJ EC00251
MOVJ C00252 BC00252 VJ=100.00  +MOVJ EC00252 VJ=100.00
MOVJ C00253 BC00253 VJ=100.00  +MOVJ EC00253 VJ=100.00
END
